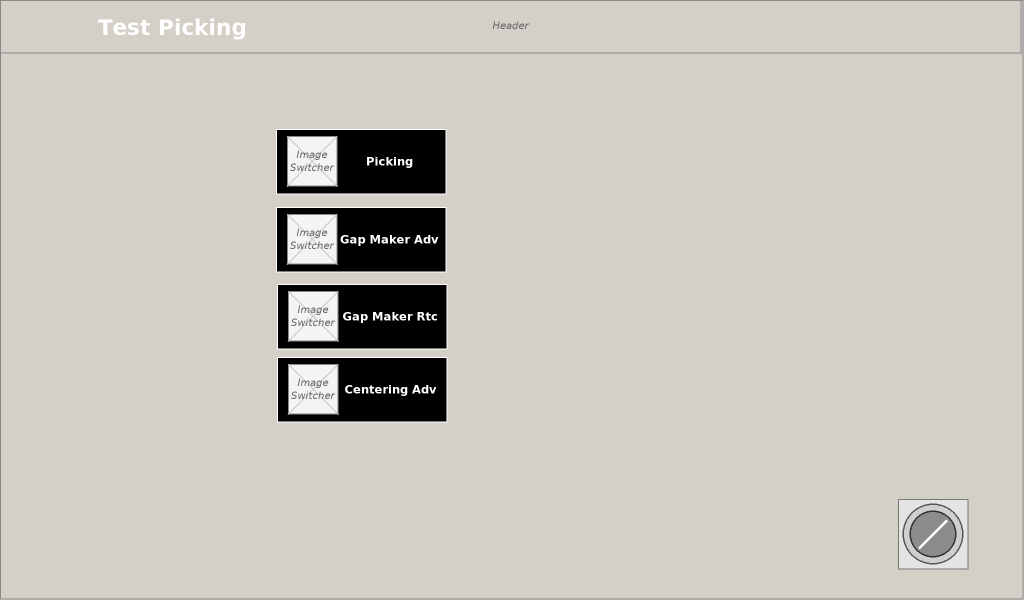
VISUALIZATION Test_Picking  // 1024x600
    Frame (0,-2 1021x55)
        shows Header()
    Label (95,15 250x25), "Test Picking"
    RotarySwitch (898,499 70x70), variable: HMI_GVL.bTestModeEnablePicking, behaviour: TOGGLE, style: Switch-RotarySwitch-Gray
    RoundedRectangle (276,129 170x65)
        toggle Status_GVL.stMotor_Picking.iTestForward
    Label (321,149 137x25), "Picking"
    ImageSwitcher (287,136 50x50), variable: Status_GVL.stMotor_Picking.iTestForward, behaviour: TOGGLE
    RoundedRectangle (276,207 170x65)
        toggle Status_GVL.stPneu_GapMaker.iTestAdvanced
    Label (321,227 137x25), "Gap Maker Adv"
    ImageSwitcher (287,214 50x50), variable: Status_GVL.stPneu_GapMaker.iTestAdvanced, behaviour: TOGGLE
    RoundedRectangle (277,284 170x65)
        toggle Status_GVL.stPneu_GapMaker.iTestRetract
    Label (322,304 137x25), "Gap Maker Rtc"
    ImageSwitcher (288,291 50x50), variable: Status_GVL.stPneu_GapMaker.iTestRetract, behaviour: TOGGLE
    RoundedRectangle (277,357 170x65)
        toggle Status_GVL.stPneu_Centering.iTest
    Label (322,377 137x25), "Centering Adv"
    ImageSwitcher (288,364 50x50), variable: Status_GVL.stPneu_GapMaker.iTestRetract, behaviour: TOGGLE
END_VISUALIZATION

(* stored: Version 1.1.0.1, ProductVersion 3.1.4024.12
   Visu Test_Picking: Id {721e2f95-e22c-4199-9435-c32a8dd9358d} *)
